(* IEC 61131-3 sources: io/src/Output, 11 files *)

(* ---- IBinOutput.st ---- *)
NAMESPACE Simatic.Ax.IO.Output

    /// Interface for binary output signal handling
    /// Defines the contract for controlling binary output signals
    /// Implementations provide methods to set, toggle, and query output state
    INTERFACE IBinOutput

        /// Set the output to a specific boolean value
        /// value: TRUE to turn output on, FALSE to turn output off
        METHOD SetQ
            VAR_INPUT
                value : BOOL;
            END_VAR
        END_METHOD

        /// Set the output to ON (TRUE)
        METHOD SetOn
        END_METHOD

        /// Set the output to OFF (FALSE)
        METHOD SetOff
        END_METHOD

        /// Toggle the output state (ON->OFF or OFF->ON)
        METHOD Toggle
        END_METHOD

        /// Returns the current state of the output
        /// RETURN: TRUE if output is on, FALSE if output is off
        METHOD IsOn : BOOL
        END_METHOD
    END_INTERFACE

    /// Null Object pattern implementation for ItfBinOutput
    /// Provides a safe default implementation that does nothing
    /// Use this to avoid null pointer checks when a binary output is optional
    CLASS NullBinOutput
        IMPLEMENTS IBinOutput

        /// Set output to specific value (no operation for null object)
        /// value: Ignored
        METHOD PUBLIC SetQ
            VAR_INPUT
                value : BOOL;
            END_VAR
            ;
        END_METHOD

        /// Set output to ON (no operation for null object)
        METHOD PUBLIC SetOn
            ;
        END_METHOD

        /// Set output to OFF (no operation for null object)
        METHOD PUBLIC SetOff
            ;
        END_METHOD

        /// Toggle output state (no operation for null object)
        METHOD PUBLIC Toggle
            ;
        END_METHOD

        /// Returns output state (always FALSE for null object)
        /// RETURN: FALSE
        METHOD PUBLIC IsOn : BOOL
            ;
        END_METHOD
    END_CLASS

END_NAMESPACE

(* ---- ItfBinOutput.st ---- *)
NAMESPACE Simatic.Ax.IO.Output

    /// Interface for binary output signal handling
    /// Defines the contract for controlling binary output signals
    /// Implementations provide methods to set, toggle, and query output state
    INTERFACE ItfBinOutput

        /// Set the output to a specific boolean value
        /// value: TRUE to turn output on, FALSE to turn output off
        METHOD SetQ
            VAR_INPUT
                value : BOOL;
            END_VAR
        END_METHOD

        /// Set the output to ON (TRUE)
        METHOD SetOn
        END_METHOD

        /// Set the output to OFF (FALSE)
        METHOD SetOff
        END_METHOD

        /// Toggle the output state (ON->OFF or OFF->ON)
        METHOD Toggle
        END_METHOD

        /// Returns the current state of the output
        /// RETURN: TRUE if output is on, FALSE if output is off
        METHOD IsOn : BOOL
        END_METHOD
    END_INTERFACE

    /// Null Object pattern implementation for ItfBinOutput
    /// Provides a safe default implementation that does nothing
    /// Use this to avoid null pointer checks when a binary output is optional
    CLASS NullBinOutput
        IMPLEMENTS ItfBinOutput

        /// Set output to specific value (no operation for null object)
        /// value: Ignored
        METHOD PUBLIC SetQ
            VAR_INPUT
                value : BOOL;
            END_VAR
            ;
        END_METHOD

        /// Set output to ON (no operation for null object)
        METHOD PUBLIC SetOn
            ;
        END_METHOD

        /// Set output to OFF (no operation for null object)
        METHOD PUBLIC SetOff
            ;
        END_METHOD

        /// Toggle output state (no operation for null object)
        METHOD PUBLIC Toggle
            ;
        END_METHOD

        /// Returns output state (always FALSE for null object)
        /// RETURN: FALSE
        METHOD PUBLIC IsOn : BOOL
            ;
        END_METHOD
    END_CLASS

END_NAMESPACE

(* ---- BinOutput.st ---- *)
NAMESPACE Simatic.Ax.IO.Output

    /// Binary output signal handler with edge detection
    /// OOP-based approach to handle digital outputs as independent objects
    /// Provides state management, edge detection (switched on/off), and change tracking
    /// Must be called cyclically via WriteCyclic() method
    CLASS BinOutput IMPLEMENTS ItfBinOutput
        VAR
            _state : BOOL;  // Internal state of the output
            _stateOld : BOOL := FALSE; // Previous state for edge detection
            _switchedOn : BOOL; // TRUE for one cycle when output switches from OFF to ON
            _switchedOff : BOOL; // TRUE for one cycle when output switches from ON to OFF
            _hasChanged : BOOL; // TRUE for one cycle when output state changes
        END_VAR

        /// Write the internal state to the digital output hardware
        /// Must be executed every cycle (recommendation: at the end of the cycle)
        /// Updates edge detection flags and outputs the current state
        /// Q: Output parameter containing the current state to be written to hardware
        METHOD PUBLIC WriteCyclic
            VAR_OUTPUT
                Q : BOOL;
            END_VAR
            // Detect edges: switched on (OFF->ON) and switched off (ON->OFF)
            _switchedOn := _state AND NOT(_stateOld);
            _switchedOff := NOT(_state) AND _stateOld;
            _hasChanged := _switchedOn OR _switchedOff;

            // Store current state for next cycle's edge detection
            _stateOld := _state;

            // Output the current state
            Q:= _state;
        END_METHOD

        /// Set the digital output to a specific boolean value
        /// value: TRUE to turn output on, FALSE to turn output off
        METHOD PUBLIC SetQ
            VAR_INPUT
                value : BOOL;
            END_VAR
            _state := value;
        END_METHOD

        /// Set the digital output to ON (TRUE)
        /// Convenience method equivalent to SetQ(TRUE)
        METHOD PUBLIC SetOn
            _state := TRUE;
        END_METHOD

        /// Set the digital output to OFF (FALSE)
        /// Convenience method equivalent to SetQ(FALSE)
        METHOD PUBLIC SetOff
            _state := FALSE;
        END_METHOD

        /// Toggle the digital output state
        /// Changes state from OFF to ON or from ON to OFF
        METHOD PUBLIC Toggle
            _state := NOT(_state);
        END_METHOD

        /// Returns the current state of the digital output
        /// RETURN: TRUE if output is on, FALSE if output is off
        METHOD PUBLIC IsOn : BOOL
            IsOn := _state;
        END_METHOD

        /// Returns TRUE if the output value has changed in the current cycle
        /// Change is detected during WriteCyclic() call
        /// RETURN: TRUE for one cycle after state change, otherwise FALSE
        METHOD PUBLIC HasChanged : BOOL
            HasChanged := _hasChanged;
        END_METHOD

        /// Returns TRUE if the output has switched on in the current cycle
        /// Switched on: transition from OFF (FALSE) to ON (TRUE)
        /// RETURN: TRUE for one cycle after switching on, otherwise FALSE
        METHOD PUBLIC HasSwitchedOn : BOOL
            HasSwitchedOn := _switchedOn;
        END_METHOD

        /// Returns TRUE if the output has switched off in the current cycle
        /// Switched off: transition from ON (TRUE) to OFF (FALSE)
        /// RETURN: TRUE for one cycle after switching off, otherwise FALSE
        METHOD PUBLIC HasSwitchedOff : BOOL
            HasSwitchedOff := _switchedOff;
        END_METHOD

    END_CLASS
END_NAMESPACE

(* ---- DintOutput.st ---- *)
NAMESPACE Simatic.Ax.IO.Output

    /// Double Integer (DINT) output signal handler with change detection
    /// Handles 32-bit signed integer output values to hardware or software targets
    /// Range: -2,147,483,648 to 2,147,483,647
    /// Provides automatic change detection when WriteCyclic() is called
    CLASS DintOutput EXTENDS OutputBase
        VAR
            _actualValue : DINT; // Current output value to be written
            _oldValue : DINT; // Previous output value for change detection
        END_VAR

        /// Set the double integer output value
        /// The value is stored internally and written during WriteCyclic() call
        /// value: DINT value to set (range: -2,147,483,648 to 2,147,483,647)
        METHOD PUBLIC SetValue
            VAR_INPUT
                value : DINT;
            END_VAR
            _actualValue := value;
        END_METHOD

        /// Write the value to the output periphery cyclically
        /// Must be executed every cycle (recommendation: at the end of the cycle)
        /// Updates change detection and outputs the current value
        /// Can also be used for non-hardware (software-only) outputs
        /// Q: Output parameter containing the current DINT value
        METHOD PUBLIC WriteCyclic
            VAR_OUTPUT
                Q : DINT;
            END_VAR
            THIS.HasChanged(value := _actualValue <> _oldValue);
            _oldValue := _actualValue;
            Q:= _actualValue;
        END_METHOD
    END_CLASS
END_NAMESPACE

(* ---- DWordOutput.st ---- *)
NAMESPACE Simatic.Ax.IO.Output

    /// Double Word (DWORD) output signal handler with change detection
    /// Handles 32-bit unsigned word output values to hardware or software targets
    /// Range: 0 (16#0) to 4,294,967,295 (16#FFFFFFFF)
    /// Typically used for bit patterns, status words, or unsigned integer values
    CLASS DWordOutput EXTENDS OutputBase
        VAR
            _actualValue : DWORD; // Current output value to be written
            _oldValue : DWORD; // Previous output value for change detection
        END_VAR

        /// Set the double word output value
        /// The value is stored internally and written during WriteCyclic() call
        /// value: DWORD value to set (range: 0 to 4,294,967,295)
        METHOD PUBLIC SetValue
            VAR_INPUT
                value : DWORD;
            END_VAR
            _actualValue := value;
        END_METHOD

        /// Write the value to the output periphery cyclically
        /// Must be executed every cycle (recommendation: at the end of the cycle)
        /// Updates change detection and outputs the current value
        /// Can also be used for non-hardware (software-only) outputs
        /// Q: Output parameter containing the current DWORD value
        METHOD PUBLIC WriteCyclic
            VAR_OUTPUT
                Q : DWORD;
            END_VAR
            THIS.HasChanged(value := _actualValue <> _oldValue);
            _oldValue := _actualValue;
            Q:= _actualValue;
        END_METHOD
    END_CLASS
END_NAMESPACE

(* ---- IntOutput.st ---- *)
NAMESPACE Simatic.Ax.IO.Output

    /// Integer (INT) output signal handler with change detection
    /// Handles 16-bit signed integer output values to hardware or software targets
    /// Range: -32768 to 32767
    /// Provides automatic change detection when WriteCyclic() is called
    CLASS IntOutput EXTENDS OutputBase
        VAR
            _actualValue : INT; // Current output value to be written
            _oldValue : INT; // Previous output value for change detection
        END_VAR

        /// Set the integer output value
        /// The value is stored internally and written during WriteCyclic() call
        /// value: INT value to set (range: -32768 to 32767)
        METHOD PUBLIC SetValue
            VAR_INPUT
                value : INT;
            END_VAR
            _actualValue := value;
        END_METHOD

        /// Write the value to the output periphery cyclically
        /// Must be executed every cycle (recommendation: at the end of the cycle)
        /// Updates change detection and outputs the current value
        /// Can also be used for non-hardware (software-only) outputs
        /// Q: Output parameter containing the current INT value
        METHOD PUBLIC WriteCyclic
            VAR_OUTPUT
                Q : INT;
            END_VAR
            THIS.HasChanged(value := _actualValue <> _oldValue);
            _oldValue := _actualValue;
            Q:= _actualValue;
        END_METHOD
    END_CLASS
END_NAMESPACE

(* ---- LIntOutput.st ---- *)
NAMESPACE Simatic.Ax.IO.Output

    /// Long Integer (LINT) output signal handler with change detection
    /// Handles 64-bit signed integer output values to hardware or software targets
    /// Range: -9,223,372,036,854,775,808 to 9,223,372,036,854,775,807
    /// Provides automatic change detection when WriteCyclic() is called
    CLASS LIntOutput EXTENDS OutputBase
        VAR
            _actualValue : LINT; // Current output value to be written
            _oldValue : LINT; // Previous output value for change detection
        END_VAR

        /// Set the long integer output value
        /// The value is stored internally and written during WriteCyclic() call
        /// value: LINT value to set (64-bit signed integer)
        METHOD PUBLIC SetValue
            VAR_INPUT
                value : LINT;
            END_VAR
            _actualValue := value;
        END_METHOD

        /// Write the value to the output periphery cyclically
        /// Must be executed every cycle (recommendation: at the end of the cycle)
        /// Updates change detection and outputs the current value
        /// Can also be used for non-hardware (software-only) outputs
        /// Q: Output parameter containing the current LINT value
        METHOD PUBLIC WriteCyclic
            VAR_OUTPUT
                Q : LINT;
            END_VAR
            THIS.HasChanged(value := _actualValue <> _oldValue);
            _oldValue := _actualValue;
            Q:= _actualValue;
        END_METHOD
    END_CLASS
END_NAMESPACE

(* ---- LRealOutput.st ---- *)
NAMESPACE Simatic.Ax.IO.Output

    /// Long Real (LREAL) floating-point output signal handler with change detection
    /// Handles 64-bit double precision floating-point output values to hardware or software targets
    /// Range: approximately ±1.8e308 (double precision IEEE 754)
    /// Outputs as LWORD bit pattern for hardware compatibility
    CLASS LRealOutput EXTENDS OutputBase
        VAR
            _actualValue : LREAL; // Current output value to be written
            _oldValue : LREAL; // Previous output value for change detection
        END_VAR

        /// Set the long real floating-point output value
        /// The value is stored internally and written during WriteCyclic() call
        /// value: LREAL value to set (64-bit double precision floating-point)
        METHOD PUBLIC SetValue
            VAR_INPUT
                value : LREAL;
            END_VAR
            _actualValue := value;
        END_METHOD

        /// Write the value to the output periphery cyclically
        /// Must be executed every cycle (recommendation: at the end of the cycle)
        /// Updates change detection and outputs the current value as LWORD bit pattern
        /// Can also be used for non-hardware (software-only) outputs
        /// Q: Output parameter containing the current LREAL value as LWORD bit pattern
        METHOD PUBLIC WriteCyclic
            VAR_OUTPUT
                Q : LWORD;
            END_VAR
            THIS.HasChanged(value := _actualValue <> _oldValue);
            _oldValue := _actualValue;
            Q:= TO_LWORD(_actualValue);
        END_METHOD

    END_CLASS
END_NAMESPACE

(* ---- OutputBase.st ---- *)
NAMESPACE Simatic.Ax.IO.Output

    /// Base class for all output signal types
    /// Provides common functionality for change detection
    /// This class should be extended by specific output type implementations
    CLASS OutputBase
        VAR
            _hasChanged : BOOL; // TRUE: value changed in the last cycle
        END_VAR

        /// Returns TRUE if the output value has changed in the last cycle
        /// Change detection is updated during WriteCyclic() calls
        /// RETURN: TRUE if value changed, FALSE if value remained the same
        METHOD PUBLIC HasChanged : BOOL
            HasChanged := _hasChanged;
        END_METHOD

        /// Set the change detection status internally
        /// Used by derived classes to indicate when output value has changed
        /// Must be called by derived classes in their WriteCyclic() method
        /// value: TRUE if the value has changed, FALSE otherwise
        METHOD PROTECTED HasChanged
            VAR_INPUT
                value : BOOL;
            END_VAR
            _hasChanged := true;
        END_METHOD

    END_CLASS
END_NAMESPACE

(* ---- RealOutput.st ---- *)
NAMESPACE Simatic.Ax.IO.Output

    /// Real (REAL) floating-point output signal handler with change detection
    /// Handles 32-bit floating-point output values to hardware or software targets
    /// Range: approximately ±3.4e38 (single precision IEEE 754)
    /// Outputs as DWORD bit pattern for hardware compatibility
    CLASS RealOutput EXTENDS OutputBase
        VAR
            _actualValue : REAL; // Current output value to be written
            _oldValue : REAL; // Previous output value for change detection
        END_VAR

        /// Set the real floating-point output value
        /// The value is stored internally and written during WriteCyclic() call
        /// value: REAL value to set (32-bit floating-point)
        METHOD PUBLIC SetValue
            VAR_INPUT
                value : REAL;
            END_VAR
            _actualValue := value;
        END_METHOD

        /// Write the value to the output periphery cyclically
        /// Must be executed every cycle (recommendation: at the end of the cycle)
        /// Updates change detection and outputs the current value as DWORD bit pattern
        /// Can also be used for non-hardware (software-only) outputs
        /// Q: Output parameter containing the current REAL value as DWORD bit pattern
        METHOD PUBLIC WriteCyclic
            VAR_OUTPUT
                Q : DWORD;
            END_VAR
            THIS.HasChanged(value := _actualValue <> _oldValue);
            _oldValue := _actualValue;
            Q:= TO_DWORD(_actualValue);
        END_METHOD

    END_CLASS
END_NAMESPACE

(* ---- WordOutput.st ---- *)
NAMESPACE Simatic.Ax.IO.Output

    /// Word (WORD) output signal handler with change detection
    /// Handles 16-bit unsigned word output values to hardware or software targets
    /// Range: 0 (16#0) to 65535 (16#FFFF)
    /// Typically used for bit patterns, status words, or unsigned integer values
    CLASS WordOutput EXTENDS OutputBase
        VAR
            _actualValue : WORD; // Current output value to be written
            _oldValue : WORD; // Previous output value for change detection
        END_VAR

        /// Set the word output value
        /// The value is stored internally and written during WriteCyclic() call
        /// value: WORD value to set (range: 0 to 65535)
        METHOD PUBLIC SetValue
            VAR_INPUT
                value : WORD;
            END_VAR
            _actualValue := value;
        END_METHOD

        /// Write the value to the output periphery cyclically
        /// Must be executed every cycle (recommendation: at the end of the cycle)
        /// Updates change detection and outputs the current value
        /// Can also be used for non-hardware (software-only) outputs
        /// Q: Output parameter containing the current WORD value
        METHOD PUBLIC WriteCyclic
            VAR_OUTPUT
                Q : WORD;
            END_VAR
            THIS.HasChanged(value := _actualValue <> _oldValue);
            _oldValue := _actualValue;
            Q:= _actualValue;
        END_METHOD
    END_CLASS
END_NAMESPACE
